// TIA Portal V18 export
FUNCTION_BLOCK "Calculations"   // FB10, LAD
{ S7_Optimized_Access := 'TRUE' }
// stored: AutoNumber false, MemoryReserve 100, SetENOAutomatically false
   VAR
      M1_LPF { S7_SetPoint := 'True'} : "LowPassFilter";
      M2_LPF { S7_SetPoint := 'True'} : "LowPassFilter";
      TDPressFwd_LPF { S7_SetPoint := 'True'} : "LowPassFilter";
      TDPressRev_LPF { S7_SetPoint := 'True'} : "LowPassFilter";
      ClosedLoopTemp_LPF { S7_SetPoint := 'True'} : "LowPassFilter";
      ChargeFlow_LPF { S7_SetPoint := 'True'} : "LowPassFilter";
      HotOilFlow_LPF { S7_SetPoint := 'True'} : "LowPassFilter";
      AuxFlow_LPF { S7_SetPoint := 'True'} : "LowPassFilter";
      ChargePress1_LPF { S7_SetPoint := 'True'} : "LowPassFilter";
      ChargePress2_LPF { S7_SetPoint := 'True'} : "LowPassFilter";
      DrillTorqPotLPF { S7_SetPoint := 'True'} : "LowPassFilter";
      MUTorqPotLPF { S7_SetPoint := 'True'} : "LowPassFilter";
      DrillThrottlePotLPF { S7_SetPoint := 'True'} : "LowPassFilter";
      ActTorq_LPF { S7_SetPoint := 'True'} : "LowPassFilter";
      DrillRecPTO_TP { S7_SetPoint := 'True'} : TP_TIME;
      DrillRecMax { S7_SetPoint := 'True'} : Bool;   // Send max value out to drill recorder
   END_VAR
   VAR_TEMP
      tempReal : Real;
      AutoMUTorqSetLow : Real;
      AutoMUTorqSetHigh : Real;
   END_VAR
   VAR_TEMP   // added for the SCL form of the ladder/FBD networks
      _w1 : Bool;
      _w2 : Bool;
      _w3 : Bool;
      _w4 : Bool;
      _w5 : Bool;
      _w6 : Bool;
   END_VAR
BEGIN

REGION Network 1: Encoder Position
   // Hard coded rollover value to match encoder rollver value from TM Count card
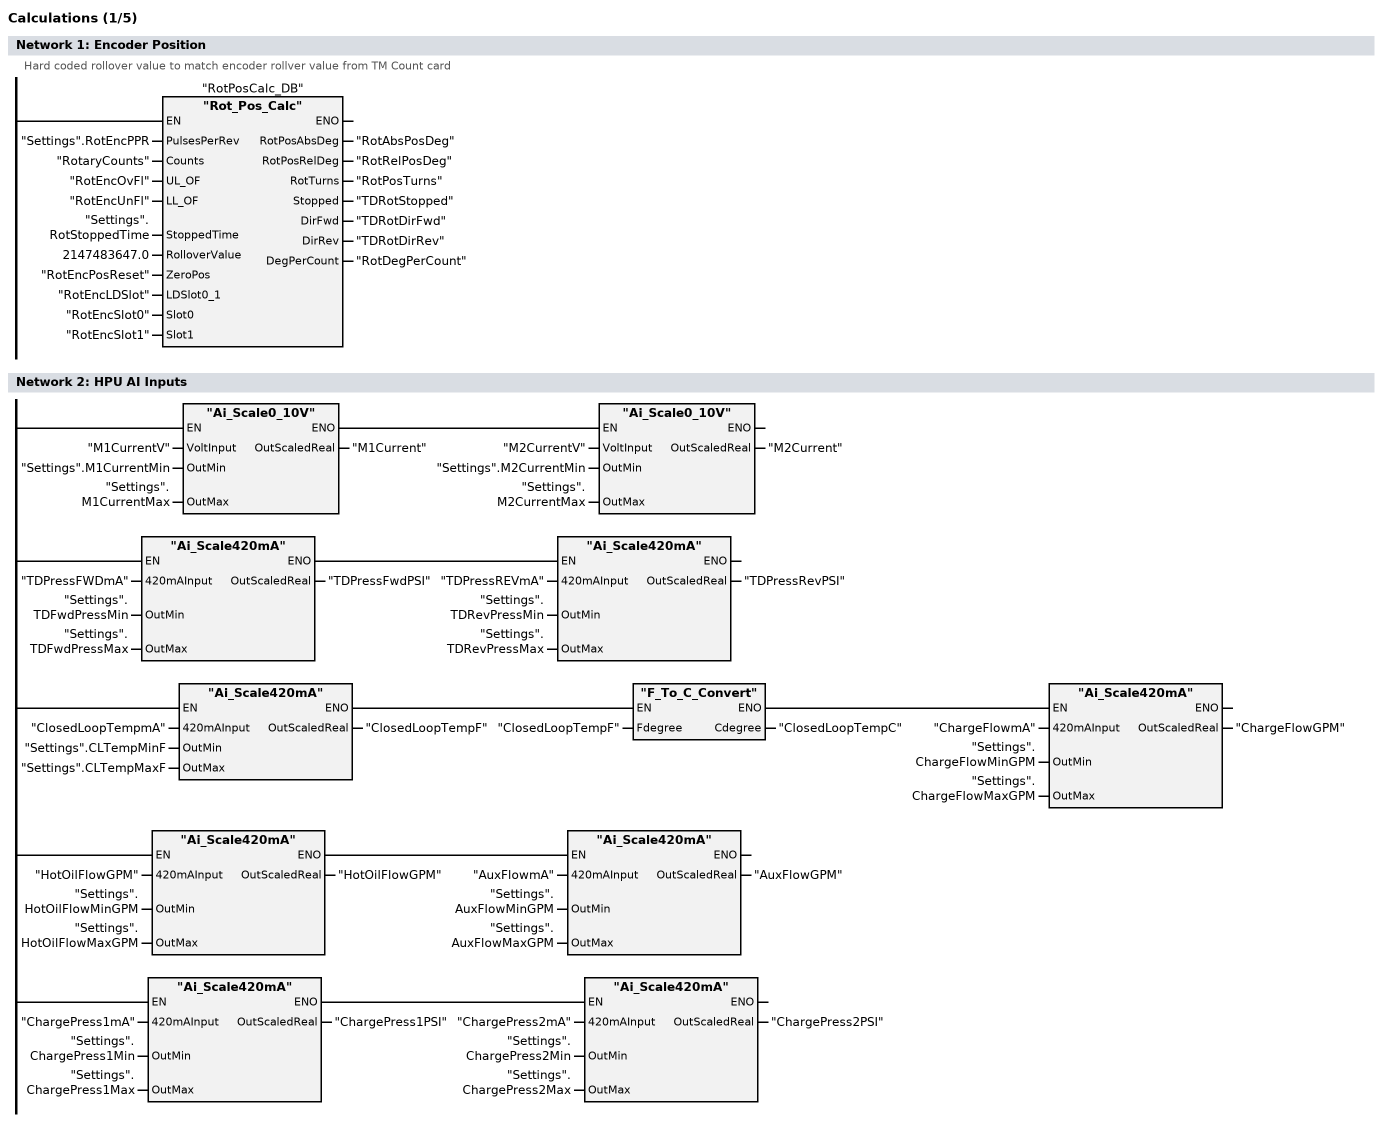
   RUNG wire#powerrail
      "RotPosCalc_DB"(PulsesPerRev := "Settings".RotEncPPR, Counts := "RotaryCounts", UL_OF := "RotEncOvFl", LL_OF := "RotEncUnFl", StoppedTime := "Settings".RotStoppedTime, RolloverValue := 2147483647.0, ZeroPos := "RotEncPosReset", LDSlot0_1 := "RotEncLDSlot", Slot0 := "RotEncSlot0", Slot1 := "RotEncSlot1", RotPosAbsDeg => "RotAbsPosDeg", RotPosRelDeg => "RotRelPosDeg", RotTurns => "RotPosTurns", Stopped => "TDRotStopped", DirFwd => "TDRotDirFwd", DirRev => "TDRotDirRev", DegPerCount => "RotDegPerCount")
   END_RUNG
   // the same network as SCL:
   "RotPosCalc_DB"(PulsesPerRev := "Settings".RotEncPPR,   // "Rot_Pos_Calc"
                   Counts := "RotaryCounts",
                   UL_OF := "RotEncOvFl",
                   LL_OF := "RotEncUnFl",
                   StoppedTime := "Settings".RotStoppedTime,
                   RolloverValue := 2147483647.0,
                   ZeroPos := "RotEncPosReset",
                   LDSlot0_1 := "RotEncLDSlot",
                   Slot0 := "RotEncSlot0",
                   Slot1 := "RotEncSlot1",
                   RotPosAbsDeg => "RotAbsPosDeg",
                   RotPosRelDeg => "RotRelPosDeg",
                   RotTurns => "RotPosTurns",
                   Stopped => "TDRotStopped",
                   DirFwd => "TDRotDirFwd",
                   DirRev => "TDRotDirRev",
                   DegPerCount => "RotDegPerCount");
END_REGION

REGION Network 2: HPU AI Inputs
   RUNG wire#powerrail
      "Ai_Scale0_10V"(VoltInput := "M1CurrentV", OutMin := "Settings".M1CurrentMin, OutMax := "Settings".M1CurrentMax, OutScaledReal => "M1Current")
      "Ai_Scale0_10V"(VoltInput := "M2CurrentV", OutMin := "Settings".M2CurrentMin, OutMax := "Settings".M2CurrentMax, OutScaledReal => "M2Current")
   END_RUNG
   RUNG wire#powerrail
      "Ai_Scale420mA"("420mAInput" := "TDPressFWDmA", OutMin := "Settings".TDFwdPressMin, OutMax := "Settings".TDFwdPressMax, OutScaledReal => "TDPressFwdPSI")
      "Ai_Scale420mA"("420mAInput" := "TDPressREVmA", OutMin := "Settings".TDRevPressMin, OutMax := "Settings".TDRevPressMax, OutScaledReal => "TDPressRevPSI")
   END_RUNG
   RUNG wire#powerrail
      "Ai_Scale420mA"("420mAInput" := "ClosedLoopTempmA", OutMin := "Settings".CLTempMinF, OutMax := "Settings".CLTempMaxF, OutScaledReal => "ClosedLoopTempF")
      "F_To_C_Convert"(Fdegree := "ClosedLoopTempF", Cdegree => "ClosedLoopTempC")
      "Ai_Scale420mA"("420mAInput" := "ChargeFlowmA", OutMin := "Settings".ChargeFlowMinGPM, OutMax := "Settings".ChargeFlowMaxGPM, OutScaledReal => "ChargeFlowGPM")
   END_RUNG
   RUNG wire#powerrail
      "Ai_Scale420mA"("420mAInput" := "HotOilFlowGPM", OutMin := "Settings".HotOilFlowMinGPM, OutMax := "Settings".HotOilFlowMaxGPM, OutScaledReal => "HotOilFlowGPM")
      "Ai_Scale420mA"("420mAInput" := "AuxFlowmA", OutMin := "Settings".AuxFlowMinGPM, OutMax := "Settings".AuxFlowMaxGPM, OutScaledReal => "AuxFlowGPM")
   END_RUNG
   RUNG wire#powerrail
      "Ai_Scale420mA"("420mAInput" := "ChargePress1mA", OutMin := "Settings".ChargePress1Min, OutMax := "Settings".ChargePress1Max, OutScaledReal => "ChargePress1PSI")
      "Ai_Scale420mA"("420mAInput" := "ChargePress2mA", OutMin := "Settings".ChargePress2Min, OutMax := "Settings".ChargePress2Max, OutScaledReal => "ChargePress2PSI")
   END_RUNG
   // the same network as SCL:
   "Ai_Scale0_10V"(VoltInput := "M1CurrentV",
                   OutMin := "Settings".M1CurrentMin,
                   OutMax := "Settings".M1CurrentMax,
                   OutScaledReal => "M1Current",
                   ENO => #_w1);
   IF #_w1 THEN
       "Ai_Scale0_10V"(VoltInput := "M2CurrentV",
                       OutMin := "Settings".M2CurrentMin,
                       OutMax := "Settings".M2CurrentMax,
                       OutScaledReal => "M2Current");
   END_IF;
   "Ai_Scale420mA"("420mAInput" := "TDPressFWDmA",
                   OutMin := "Settings".TDFwdPressMin,
                   OutMax := "Settings".TDFwdPressMax,
                   OutScaledReal => "TDPressFwdPSI",
                   ENO => #_w2);
   IF #_w2 THEN
       "Ai_Scale420mA"("420mAInput" := "TDPressREVmA",
                       OutMin := "Settings".TDRevPressMin,
                       OutMax := "Settings".TDRevPressMax,
                       OutScaledReal => "TDPressRevPSI");
   END_IF;
   "Ai_Scale420mA"("420mAInput" := "ClosedLoopTempmA",
                   OutMin := "Settings".CLTempMinF,
                   OutMax := "Settings".CLTempMaxF,
                   OutScaledReal => "ClosedLoopTempF",
                   ENO => #_w3);
   "F_To_C_Convert"(EN := #_w3, Fdegree := "ClosedLoopTempF", Cdegree => "ClosedLoopTempC", ENO => #_w4);
   IF #_w4 THEN
       "Ai_Scale420mA"("420mAInput" := "ChargeFlowmA",
                       OutMin := "Settings".ChargeFlowMinGPM,
                       OutMax := "Settings".ChargeFlowMaxGPM,
                       OutScaledReal => "ChargeFlowGPM");
   END_IF;
   "Ai_Scale420mA"("420mAInput" := "HotOilFlowGPM",
                   OutMin := "Settings".HotOilFlowMinGPM,
                   OutMax := "Settings".HotOilFlowMaxGPM,
                   OutScaledReal => "HotOilFlowGPM",
                   ENO => #_w5);
   IF #_w5 THEN
       "Ai_Scale420mA"("420mAInput" := "AuxFlowmA",
                       OutMin := "Settings".AuxFlowMinGPM,
                       OutMax := "Settings".AuxFlowMaxGPM,
                       OutScaledReal => "AuxFlowGPM");
   END_IF;
   "Ai_Scale420mA"("420mAInput" := "ChargePress1mA",
                   OutMin := "Settings".ChargePress1Min,
                   OutMax := "Settings".ChargePress1Max,
                   OutScaledReal => "ChargePress1PSI",
                   ENO => #_w6);
   IF #_w6 THEN
       "Ai_Scale420mA"("420mAInput" := "ChargePress2mA",
                       OutMin := "Settings".ChargePress2Min,
                       OutMax := "Settings".ChargePress2Max,
                       OutScaledReal => "ChargePress2PSI");
   END_IF;
END_REGION

REGION Network 3: Filter HPU Inputs
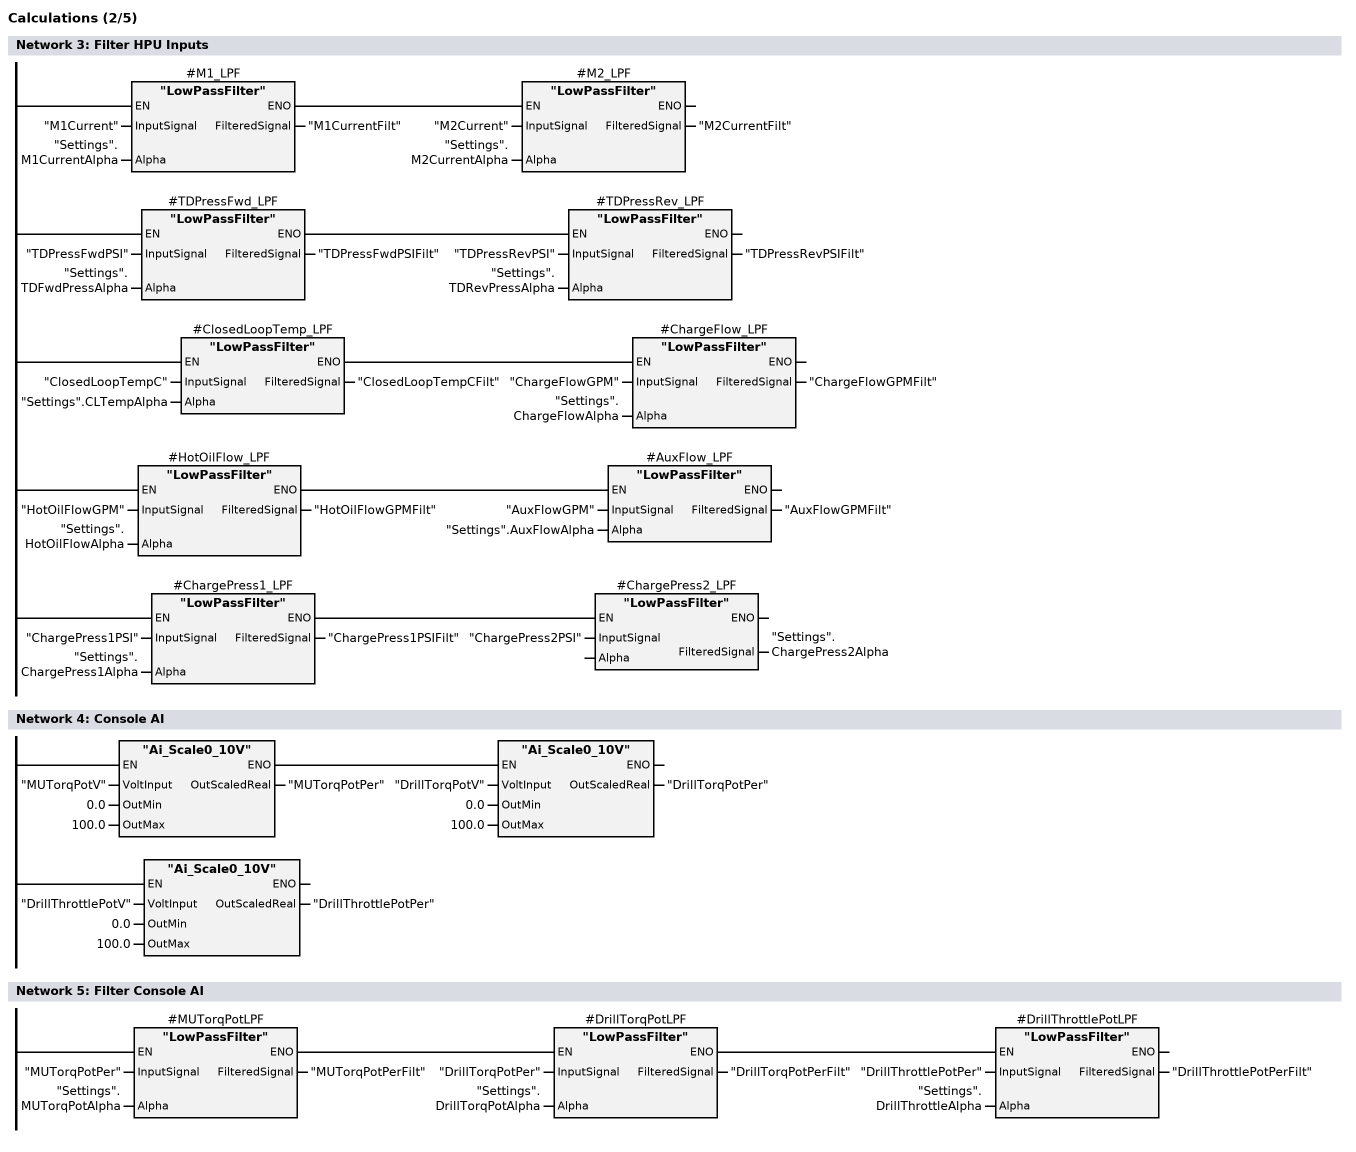
   RUNG wire#powerrail
      #M1_LPF(InputSignal := "M1Current", Alpha := "Settings".M1CurrentAlpha, FilteredSignal => "M1CurrentFilt")
      #M2_LPF(InputSignal := "M2Current", Alpha := "Settings".M2CurrentAlpha, FilteredSignal => "M2CurrentFilt")
   END_RUNG
   RUNG wire#powerrail
      #TDPressFwd_LPF(InputSignal := "TDPressFwdPSI", Alpha := "Settings".TDFwdPressAlpha, FilteredSignal => "TDPressFwdPSIFilt")
      #TDPressRev_LPF(InputSignal := "TDPressRevPSI", Alpha := "Settings".TDRevPressAlpha, FilteredSignal => "TDPressRevPSIFilt")
   END_RUNG
   RUNG wire#powerrail
      #ClosedLoopTemp_LPF(InputSignal := "ClosedLoopTempC", Alpha := "Settings".CLTempAlpha, FilteredSignal => "ClosedLoopTempCFilt")
      #ChargeFlow_LPF(InputSignal := "ChargeFlowGPM", Alpha := "Settings".ChargeFlowAlpha, FilteredSignal => "ChargeFlowGPMFilt")
   END_RUNG
   RUNG wire#powerrail
      #HotOilFlow_LPF(InputSignal := "HotOilFlowGPM", Alpha := "Settings".HotOilFlowAlpha, FilteredSignal => "HotOilFlowGPMFilt")
      #AuxFlow_LPF(InputSignal := "AuxFlowGPM", Alpha := "Settings".AuxFlowAlpha, FilteredSignal => "AuxFlowGPMFilt")
   END_RUNG
   RUNG wire#powerrail
      #ChargePress1_LPF(InputSignal := "ChargePress1PSI", Alpha := "Settings".ChargePress1Alpha, FilteredSignal => "ChargePress1PSIFilt")
      #ChargePress2_LPF(InputSignal := "ChargePress2PSI", Alpha :=, FilteredSignal => "Settings".ChargePress2Alpha)
   END_RUNG
   // the same network as SCL:
   #M1_LPF(InputSignal := "M1Current",   // "LowPassFilter"
           Alpha := "Settings".M1CurrentAlpha,
           FilteredSignal => "M1CurrentFilt",
           ENO => #_w1);
   IF #_w1 THEN
       #M2_LPF(InputSignal := "M2Current", Alpha := "Settings".M2CurrentAlpha, FilteredSignal => "M2CurrentFilt");   // "LowPassFilter"
   END_IF;
   #TDPressFwd_LPF(InputSignal := "TDPressFwdPSI",   // "LowPassFilter"
                   Alpha := "Settings".TDFwdPressAlpha,
                   FilteredSignal => "TDPressFwdPSIFilt",
                   ENO => #_w2);
   IF #_w2 THEN
       #TDPressRev_LPF(InputSignal := "TDPressRevPSI",   // "LowPassFilter"
                       Alpha := "Settings".TDRevPressAlpha,
                       FilteredSignal => "TDPressRevPSIFilt");
   END_IF;
   #ClosedLoopTemp_LPF(InputSignal := "ClosedLoopTempC",   // "LowPassFilter"
                       Alpha := "Settings".CLTempAlpha,
                       FilteredSignal => "ClosedLoopTempCFilt",
                       ENO => #_w3);
   IF #_w3 THEN
       #ChargeFlow_LPF(InputSignal := "ChargeFlowGPM",   // "LowPassFilter"
                       Alpha := "Settings".ChargeFlowAlpha,
                       FilteredSignal => "ChargeFlowGPMFilt");
   END_IF;
   #HotOilFlow_LPF(InputSignal := "HotOilFlowGPM",   // "LowPassFilter"
                   Alpha := "Settings".HotOilFlowAlpha,
                   FilteredSignal => "HotOilFlowGPMFilt",
                   ENO => #_w4);
   IF #_w4 THEN
       #AuxFlow_LPF(InputSignal := "AuxFlowGPM",   // "LowPassFilter"
                    Alpha := "Settings".AuxFlowAlpha,
                    FilteredSignal => "AuxFlowGPMFilt");
   END_IF;
   #ChargePress1_LPF(InputSignal := "ChargePress1PSI",   // "LowPassFilter"
                     Alpha := "Settings".ChargePress1Alpha,
                     FilteredSignal => "ChargePress1PSIFilt",
                     ENO => #_w5);
   IF #_w5 THEN
       #ChargePress2_LPF(InputSignal := "ChargePress2PSI", FilteredSignal => "Settings".ChargePress2Alpha);   // "LowPassFilter"
   END_IF;
END_REGION

REGION Network 4: Console AI
   RUNG wire#powerrail
      "Ai_Scale0_10V"(VoltInput := "MUTorqPotV", OutMin := 0.0, OutMax := 100.0, OutScaledReal => "MUTorqPotPer")
      "Ai_Scale0_10V"(VoltInput := "DrillTorqPotV", OutMin := 0.0, OutMax := 100.0, OutScaledReal => "DrillTorqPotPer")
   END_RUNG
   RUNG wire#powerrail
      "Ai_Scale0_10V"(VoltInput := "DrillThrottlePotV", OutMin := 0.0, OutMax := 100.0, OutScaledReal => "DrillThrottlePotPer")
   END_RUNG
   // the same network as SCL:
   "Ai_Scale0_10V"(VoltInput := "MUTorqPotV",
                   OutMin := 0.0,
                   OutMax := 100.0,
                   OutScaledReal => "MUTorqPotPer",
                   ENO => #_w1);
   IF #_w1 THEN
       "Ai_Scale0_10V"(VoltInput := "DrillTorqPotV",
                       OutMin := 0.0,
                       OutMax := 100.0,
                       OutScaledReal => "DrillTorqPotPer");
   END_IF;
   "Ai_Scale0_10V"(VoltInput := "DrillThrottlePotV",
                   OutMin := 0.0,
                   OutMax := 100.0,
                   OutScaledReal => "DrillThrottlePotPer");
END_REGION

REGION Network 5: Filter Console AI
   RUNG wire#powerrail
      #MUTorqPotLPF(InputSignal := "MUTorqPotPer", Alpha := "Settings".MUTorqPotAlpha, FilteredSignal => "MUTorqPotPerFilt")
      #DrillTorqPotLPF(InputSignal := "DrillTorqPotPer", Alpha := "Settings".DrillTorqPotAlpha, FilteredSignal => "DrillTorqPotPerFilt")
      #DrillThrottlePotLPF(InputSignal := "DrillThrottlePotPer", Alpha := "Settings".DrillThrottleAlpha, FilteredSignal => "DrillThrottlePotPerFilt")
   END_RUNG
   // the same network as SCL:
   #MUTorqPotLPF(InputSignal := "MUTorqPotPer",   // "LowPassFilter"
                 Alpha := "Settings".MUTorqPotAlpha,
                 FilteredSignal => "MUTorqPotPerFilt",
                 ENO => #_w1);
   #DrillTorqPotLPF(EN := #_w1,   // "LowPassFilter"
                    InputSignal := "DrillTorqPotPer",
                    Alpha := "Settings".DrillTorqPotAlpha,
                    FilteredSignal => "DrillTorqPotPerFilt",
                    ENO => #_w2);
   IF #_w2 THEN
       #DrillThrottlePotLPF(InputSignal := "DrillThrottlePotPer",   // "LowPassFilter"
                            Alpha := "Settings".DrillThrottleAlpha,
                            FilteredSignal => "DrillThrottlePotPerFilt");
   END_IF;
END_REGION

REGION Network 6: Torque Calculation
   // Differential Pressure x torque factor(ft-lbs/psi) unless bypass running * efficiency. Use raw reading value and filter after
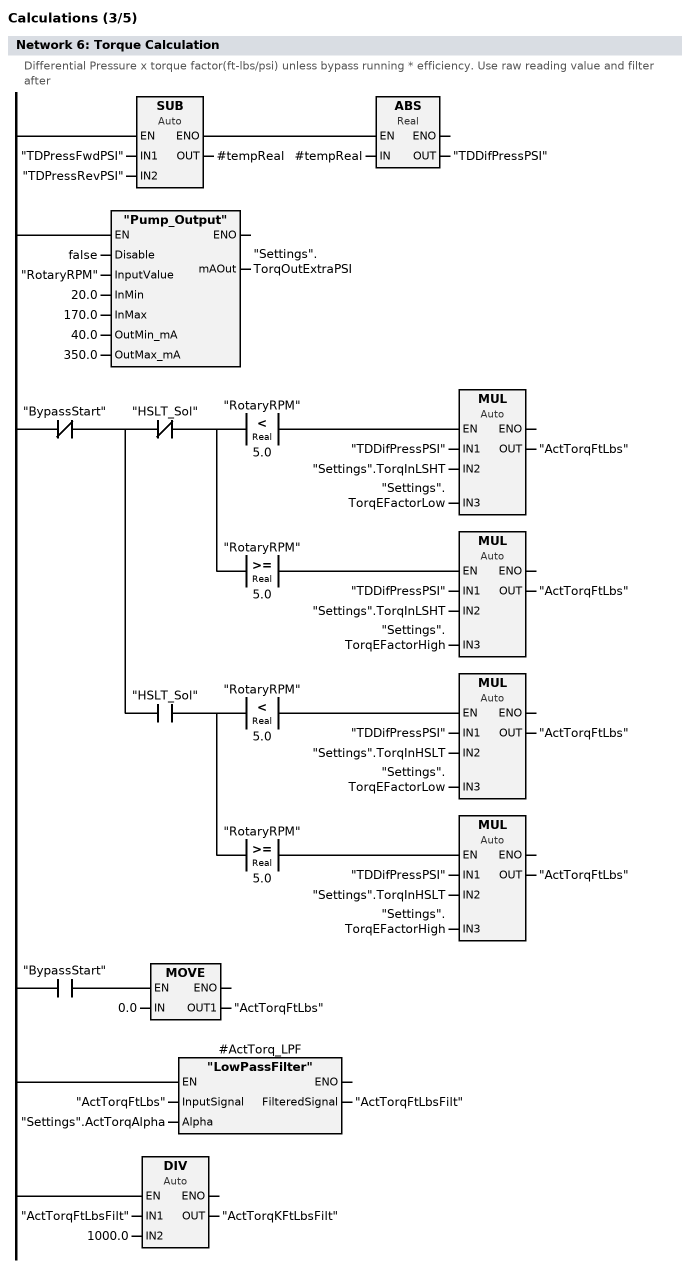
   RUNG wire#powerrail
      Sub(in1 := "TDPressFwdPSI", in2 := "TDPressRevPSI", out => #tempReal)
      { S7_Templates := "SrcType := Real" } Abs(in := #tempReal, out => "TDDifPressPSI")
   END_RUNG
   RUNG wire#powerrail
      "Pump_Output"(Disable := false, InputValue := "RotaryRPM", InMin := 20.0, InMax := 170.0, OutMin_mA := 40.0, OutMax_mA := 350.0, mAOut => "Settings".TorqOutExtraPSI)
   END_RUNG
   RUNG wire#powerrail
      I_Contact( "BypassStart" )
      wire#w1
      I_Contact( "HSLT_Sol" )
      wire#w2
      { S7_Templates := "SrcType := Real" } LT_Contact(in1 := "RotaryRPM", in2 := 5.0)
      Mul(in1 := "TDDifPressPSI", in2 := "Settings".TorqInLSHT, in3 := "Settings".TorqEFactorLow, out => "ActTorqFtLbs")
   END_RUNG
   RUNG wire#w2
      { S7_Templates := "SrcType := Real" } GE_Contact(in1 := "RotaryRPM", in2 := 5.0)
      Mul(in1 := "TDDifPressPSI", in2 := "Settings".TorqInLSHT, in3 := "Settings".TorqEFactorHigh, out => "ActTorqFtLbs")
   END_RUNG
   RUNG wire#w1
      Contact( "HSLT_Sol" )
      wire#w3
      { S7_Templates := "SrcType := Real" } LT_Contact(in1 := "RotaryRPM", in2 := 5.0)
      Mul(in1 := "TDDifPressPSI", in2 := "Settings".TorqInHSLT, in3 := "Settings".TorqEFactorLow, out => "ActTorqFtLbs")
   END_RUNG
   RUNG wire#w3
      { S7_Templates := "SrcType := Real" } GE_Contact(in1 := "RotaryRPM", in2 := 5.0)
      Mul(in1 := "TDDifPressPSI", in2 := "Settings".TorqInHSLT, in3 := "Settings".TorqEFactorHigh, out => "ActTorqFtLbs")
   END_RUNG
   RUNG wire#powerrail
      Contact( "BypassStart" )
      Move(in := 0.0, out1 => "ActTorqFtLbs")
   END_RUNG
   RUNG wire#powerrail
      #ActTorq_LPF(InputSignal := "ActTorqFtLbs", Alpha := "Settings".ActTorqAlpha, FilteredSignal => "ActTorqFtLbsFilt")
   END_RUNG
   RUNG wire#powerrail
      Div(in1 := "ActTorqFtLbsFilt", in2 := 1000.0, out => "ActTorqKFtLbsFilt")
   END_RUNG
   // the same network as SCL:
   #tempReal := "TDPressFwdPSI" - "TDPressRevPSI";
   "TDDifPressPSI" := ABS(#tempReal);
   "Pump_Output"(Disable := false,
                 InputValue := "RotaryRPM",
                 InMin := 20.0,
                 InMax := 170.0,
                 OutMin_mA := 40.0,
                 OutMax_mA := 350.0,
                 mAOut => "Settings".TorqOutExtraPSI);
   #_w1 := NOT "BypassStart" AND NOT "HSLT_Sol";
   IF #_w1 AND ("RotaryRPM" < 5.0) THEN
       "ActTorqFtLbs" := "TDDifPressPSI" * "Settings".TorqInLSHT * "Settings".TorqEFactorLow;
   END_IF;
   IF #_w1 AND ("RotaryRPM" >= 5.0) THEN
       "ActTorqFtLbs" := "TDDifPressPSI" * "Settings".TorqInLSHT * "Settings".TorqEFactorHigh;
   END_IF;
   #_w2 := NOT "BypassStart" AND "HSLT_Sol";
   IF #_w2 AND ("RotaryRPM" < 5.0) THEN
       "ActTorqFtLbs" := "TDDifPressPSI" * "Settings".TorqInHSLT * "Settings".TorqEFactorLow;
   END_IF;
   IF #_w2 AND ("RotaryRPM" >= 5.0) THEN
       "ActTorqFtLbs" := "TDDifPressPSI" * "Settings".TorqInHSLT * "Settings".TorqEFactorHigh;
   END_IF;
   IF "BypassStart" THEN "ActTorqFtLbs" := 0.0; END_IF;
   #ActTorq_LPF(InputSignal := "ActTorqFtLbs",   // "LowPassFilter"
                Alpha := "Settings".ActTorqAlpha,
                FilteredSignal => "ActTorqFtLbsFilt");
   "ActTorqKFtLbsFilt" := "ActTorqFtLbsFilt" / 1000.0;
END_REGION

REGION Network 7: User Setpoints
   // Drill torque setpoint cannot be greater than 0.95 % of the makeup setpoint
   // MU Torque always low speed as it cannot shift
   // Drill torque depends on speed settings
   // MU threshold is a percent of setpoint
   // Add 500 PSI to setpoint to overcome charge pressure
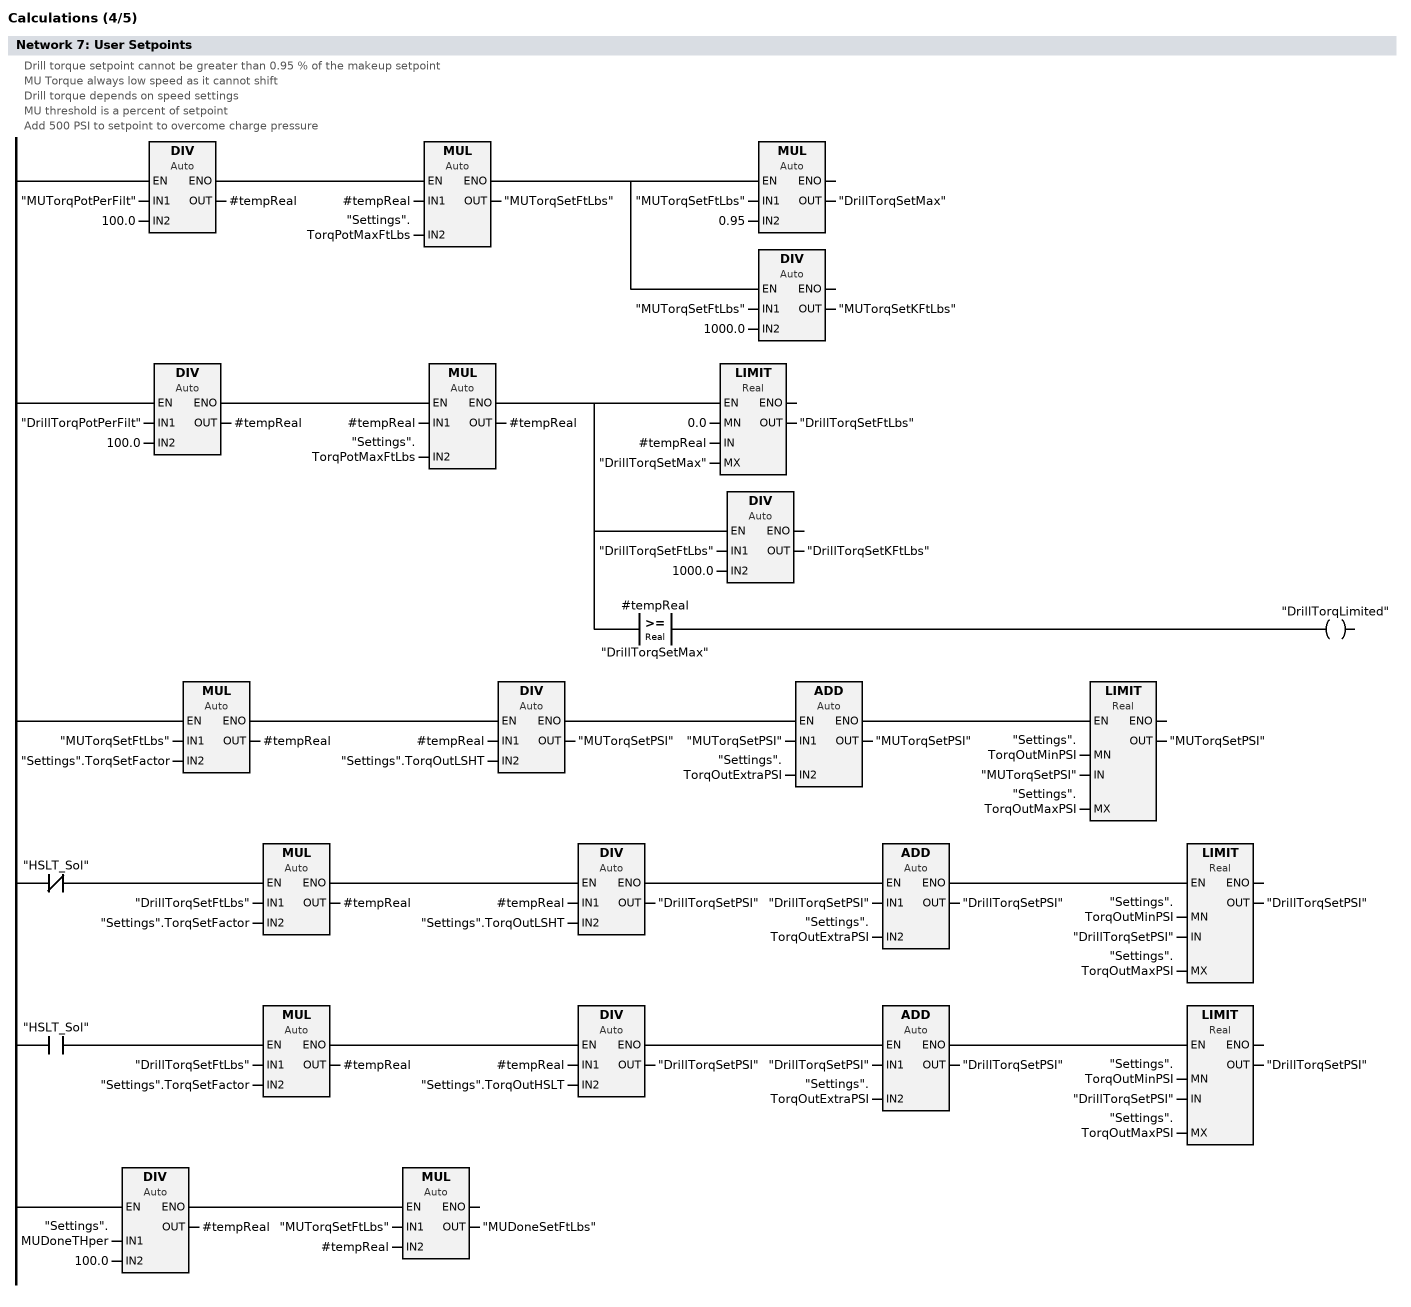
   RUNG wire#powerrail
      Div(in1 := "MUTorqPotPerFilt", in2 := 100.0, out => #tempReal)
      Mul(in1 := #tempReal, in2 := "Settings".TorqPotMaxFtLbs, out => "MUTorqSetFtLbs")
      wire#w1
      Mul(in1 := "MUTorqSetFtLbs", in2 := 0.95, out => "DrillTorqSetMax")
   END_RUNG
   RUNG wire#w1
      Div(in1 := "MUTorqSetFtLbs", in2 := 1000.0, out => "MUTorqSetKFtLbs")
   END_RUNG
   RUNG wire#powerrail
      Div(in1 := "DrillTorqPotPerFilt", in2 := 100.0, out => #tempReal)
      Mul(in1 := #tempReal, in2 := "Settings".TorqPotMaxFtLbs, out => #tempReal)
      wire#w2
      { S7_Templates := "value_type := Real" } Limit(mn := 0.0, in := #tempReal, mx := "DrillTorqSetMax", out => "DrillTorqSetFtLbs")
   END_RUNG
   RUNG wire#w2
      Div(in1 := "DrillTorqSetFtLbs", in2 := 1000.0, out => "DrillTorqSetKFtLbs")
   END_RUNG
   RUNG wire#w2
      { S7_Templates := "SrcType := Real" } GE_Contact(in1 := #tempReal, in2 := "DrillTorqSetMax")
      Coil( "DrillTorqLimited" )
   END_RUNG
   RUNG wire#powerrail
      Mul(in1 := "MUTorqSetFtLbs", in2 := "Settings".TorqSetFactor, out => #tempReal)
      Div(in1 := #tempReal, in2 := "Settings".TorqOutLSHT, out => "MUTorqSetPSI")
      Add(in1 := "MUTorqSetPSI", in2 := "Settings".TorqOutExtraPSI, out => "MUTorqSetPSI")
      { S7_Templates := "value_type := Real" } Limit(mn := "Settings".TorqOutMinPSI, in := "MUTorqSetPSI", mx := "Settings".TorqOutMaxPSI, out => "MUTorqSetPSI")
   END_RUNG
   RUNG wire#powerrail
      I_Contact( "HSLT_Sol" )
      Mul(in1 := "DrillTorqSetFtLbs", in2 := "Settings".TorqSetFactor, out => #tempReal)
      Div(in1 := #tempReal, in2 := "Settings".TorqOutLSHT, out => "DrillTorqSetPSI")
      Add(in1 := "DrillTorqSetPSI", in2 := "Settings".TorqOutExtraPSI, out => "DrillTorqSetPSI")
      { S7_Templates := "value_type := Real" } Limit(mn := "Settings".TorqOutMinPSI, in := "DrillTorqSetPSI", mx := "Settings".TorqOutMaxPSI, out => "DrillTorqSetPSI")
   END_RUNG
   RUNG wire#powerrail
      Contact( "HSLT_Sol" )
      Mul(in1 := "DrillTorqSetFtLbs", in2 := "Settings".TorqSetFactor, out => #tempReal)
      Div(in1 := #tempReal, in2 := "Settings".TorqOutHSLT, out => "DrillTorqSetPSI")
      Add(in1 := "DrillTorqSetPSI", in2 := "Settings".TorqOutExtraPSI, out => "DrillTorqSetPSI")
      { S7_Templates := "value_type := Real" } Limit(mn := "Settings".TorqOutMinPSI, in := "DrillTorqSetPSI", mx := "Settings".TorqOutMaxPSI, out => "DrillTorqSetPSI")
   END_RUNG
   RUNG wire#powerrail
      Div(in1 := "Settings".MUDoneTHper, in2 := 100.0, out => #tempReal)
      Mul(in1 := "MUTorqSetFtLbs", in2 := #tempReal, out => "MUDoneSetFtLbs")
   END_RUNG
   // the same network as SCL:
   #tempReal := "MUTorqPotPerFilt" / 100.0;
   "MUTorqSetFtLbs" := #tempReal * "Settings".TorqPotMaxFtLbs;
   "DrillTorqSetMax" := "MUTorqSetFtLbs" * 0.95;
   "MUTorqSetKFtLbs" := "MUTorqSetFtLbs" / 1000.0;
   #tempReal := "DrillTorqPotPerFilt" / 100.0;
   #tempReal := #tempReal * "Settings".TorqPotMaxFtLbs;
   "DrillTorqSetFtLbs" := LIMIT(MN := 0.0, IN := #tempReal, MX := "DrillTorqSetMax");
   "DrillTorqSetKFtLbs" := "DrillTorqSetFtLbs" / 1000.0;
   "DrillTorqLimited" := #tempReal >= "DrillTorqSetMax";
   #tempReal := "MUTorqSetFtLbs" * "Settings".TorqSetFactor;
   "MUTorqSetPSI" := #tempReal / "Settings".TorqOutLSHT;
   "MUTorqSetPSI" := "MUTorqSetPSI" + "Settings".TorqOutExtraPSI;
   "MUTorqSetPSI" := LIMIT(MN := "Settings".TorqOutMinPSI, IN := "MUTorqSetPSI", MX := "Settings".TorqOutMaxPSI);
   IF NOT "HSLT_Sol" THEN
       #tempReal := "DrillTorqSetFtLbs" * "Settings".TorqSetFactor;
       "DrillTorqSetPSI" := #tempReal / "Settings".TorqOutLSHT;
       "DrillTorqSetPSI" := "DrillTorqSetPSI" + "Settings".TorqOutExtraPSI;
       "DrillTorqSetPSI" := LIMIT(MN := "Settings".TorqOutMinPSI, IN := "DrillTorqSetPSI", MX := "Settings".TorqOutMaxPSI);
   END_IF;
   IF "HSLT_Sol" THEN
       #tempReal := "DrillTorqSetFtLbs" * "Settings".TorqSetFactor;
       "DrillTorqSetPSI" := #tempReal / "Settings".TorqOutHSLT;
       "DrillTorqSetPSI" := "DrillTorqSetPSI" + "Settings".TorqOutExtraPSI;
       "DrillTorqSetPSI" := LIMIT(MN := "Settings".TorqOutMinPSI, IN := "DrillTorqSetPSI", MX := "Settings".TorqOutMaxPSI);
   END_IF;
   #tempReal := "Settings".MUDoneTHper / 100.0;
   "MUDoneSetFtLbs" := "MUTorqSetFtLbs" * #tempReal;
END_REGION

REGION Network 8: Auto Makeup Torq Setpoints
   // These setpoints are based on a percent of the user input
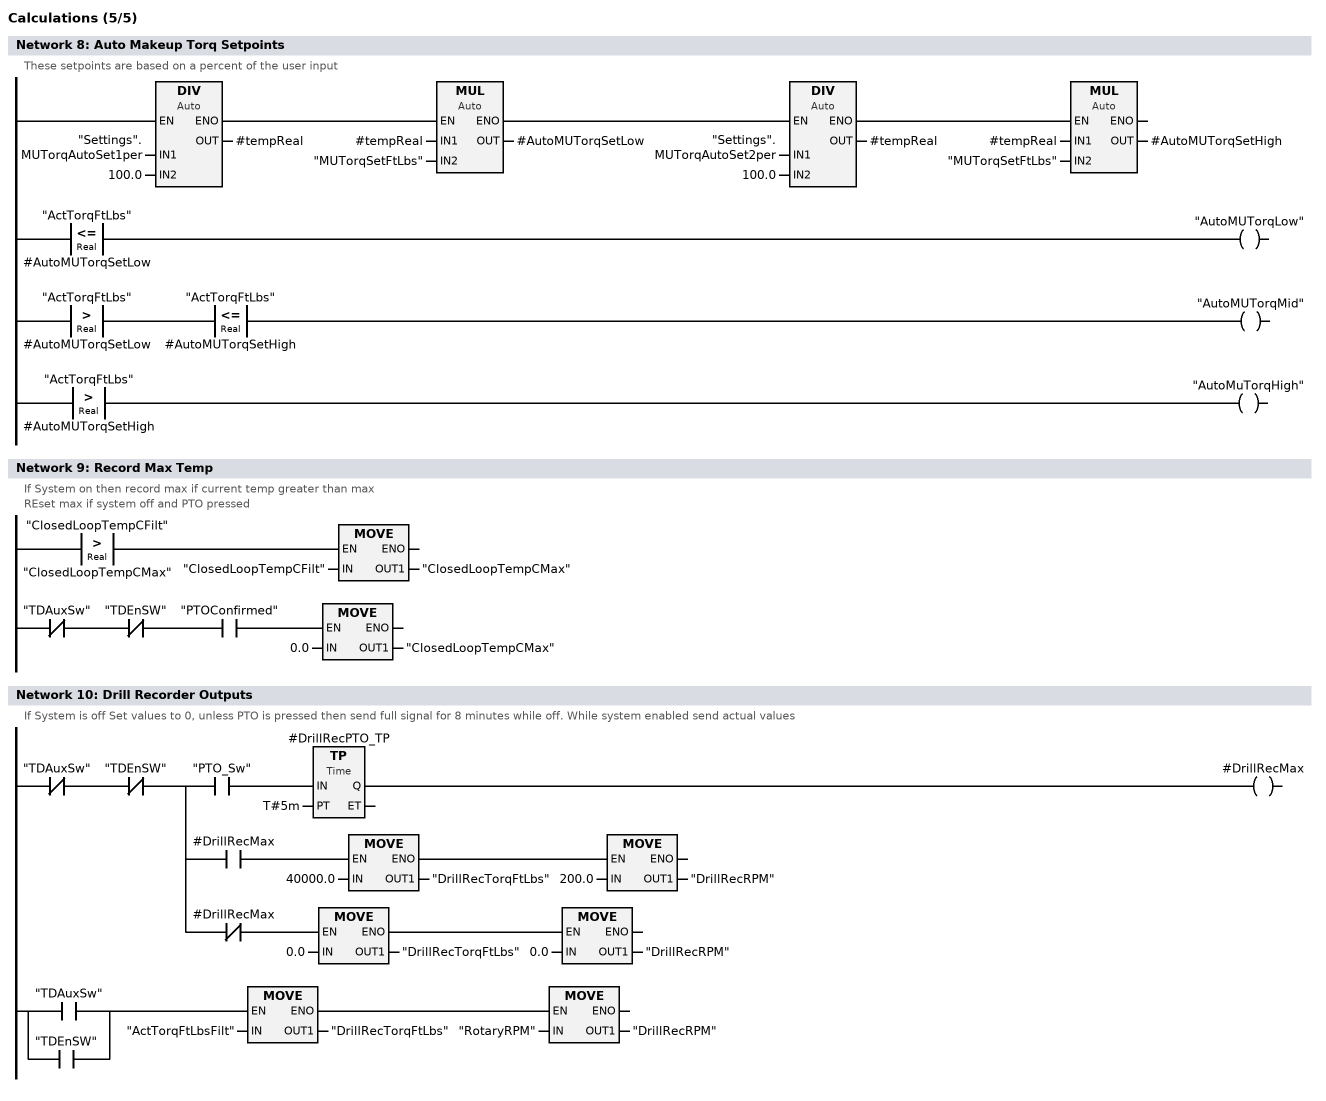
   RUNG wire#powerrail
      Div(in1 := "Settings".MUTorqAutoSet1per, in2 := 100.0, out => #tempReal)
      Mul(in1 := #tempReal, in2 := "MUTorqSetFtLbs", out => #AutoMUTorqSetLow)
      Div(in1 := "Settings".MUTorqAutoSet2per, in2 := 100.0, out => #tempReal)
      Mul(in1 := #tempReal, in2 := "MUTorqSetFtLbs", out => #AutoMUTorqSetHigh)
   END_RUNG
   RUNG wire#powerrail
      { S7_Templates := "SrcType := Real" } LE_Contact(in1 := "ActTorqFtLbs", in2 := #AutoMUTorqSetLow)
      Coil( "AutoMUTorqLow" )
   END_RUNG
   RUNG wire#powerrail
      { S7_Templates := "SrcType := Real" } GT_Contact(in1 := "ActTorqFtLbs", in2 := #AutoMUTorqSetLow)
      { S7_Templates := "SrcType := Real" } LE_Contact(in1 := "ActTorqFtLbs", in2 := #AutoMUTorqSetHigh)
      Coil( "AutoMUTorqMid" )
   END_RUNG
   RUNG wire#powerrail
      { S7_Templates := "SrcType := Real" } GT_Contact(in1 := "ActTorqFtLbs", in2 := #AutoMUTorqSetHigh)
      Coil( "AutoMuTorqHigh" )
   END_RUNG
   // the same network as SCL:
   #tempReal := "Settings".MUTorqAutoSet1per / 100.0;
   #AutoMUTorqSetLow := #tempReal * "MUTorqSetFtLbs";
   #tempReal := "Settings".MUTorqAutoSet2per / 100.0;
   #AutoMUTorqSetHigh := #tempReal * "MUTorqSetFtLbs";
   "AutoMUTorqLow" := "ActTorqFtLbs" <= #AutoMUTorqSetLow;
   "AutoMUTorqMid" := ("ActTorqFtLbs" > #AutoMUTorqSetLow) AND ("ActTorqFtLbs" <= #AutoMUTorqSetHigh);
   "AutoMuTorqHigh" := "ActTorqFtLbs" > #AutoMUTorqSetHigh;
END_REGION

REGION Network 9: Record Max Temp
   // If System on then record max if current temp greater than max
   // REset max if system off and PTO pressed
   RUNG wire#powerrail
      { S7_Templates := "SrcType := Real" } GT_Contact(in1 := "ClosedLoopTempCFilt", in2 := "ClosedLoopTempCMax")
      Move(in := "ClosedLoopTempCFilt", out1 => "ClosedLoopTempCMax")
   END_RUNG
   RUNG wire#powerrail
      I_Contact( "TDAuxSw" )
      I_Contact( "TDEnSW" )
      Contact( "PTOConfirmed" )
      Move(in := 0.0, out1 => "ClosedLoopTempCMax")
   END_RUNG
   // the same network as SCL:
   IF "ClosedLoopTempCFilt" > "ClosedLoopTempCMax" THEN
       "ClosedLoopTempCMax" := "ClosedLoopTempCFilt";
   END_IF;
   IF NOT "TDAuxSw" AND NOT "TDEnSW" AND "PTOConfirmed" THEN "ClosedLoopTempCMax" := 0.0; END_IF;
END_REGION

REGION Network 10: Drill Recorder Outputs
   // If System is off Set values to 0, unless PTO is pressed then send full signal for 8 minutes while off. While system enabled send actual values
   RUNG wire#powerrail
      I_Contact( "TDAuxSw" )
      I_Contact( "TDEnSW" )
      wire#w1
      Contact( "PTO_Sw" )
      { S7_Templates := "time_type := Time" } #DrillRecPTO_TP.TP(pt := T#5m, et =>)
      Coil( #DrillRecMax )
   END_RUNG
   RUNG wire#w1
      Contact( #DrillRecMax )
      Move(in := 40000.0, out1 => "DrillRecTorqFtLbs")
      Move(in := 200.0, out1 => "DrillRecRPM")
   END_RUNG
   RUNG wire#w1
      I_Contact( #DrillRecMax )
      Move(in := 0.0, out1 => "DrillRecTorqFtLbs")
      Move(in := 0.0, out1 => "DrillRecRPM")
   END_RUNG
   RUNG wire#powerrail
      Contact( "TDAuxSw" )
      wire#w2
      Move(in := "ActTorqFtLbsFilt", out1 => "DrillRecTorqFtLbs")
      Move(in := "RotaryRPM", out1 => "DrillRecRPM")
   END_RUNG
   RUNG wire#powerrail
      Contact( "TDEnSW" )
   END_RUNG wire#w2
   // the same network as SCL:
   #_w1 := NOT "TDAuxSw" AND NOT "TDEnSW";
   #DrillRecPTO_TP(IN := #_w1 AND "PTO_Sw", PT := T#5m);   // TP
   #DrillRecMax := #DrillRecPTO_TP.Q;
   IF #_w1 AND #DrillRecMax THEN
       "DrillRecTorqFtLbs" := 40000.0;
       "DrillRecRPM" := 200.0;
   END_IF;
   IF #_w1 AND NOT #DrillRecMax THEN
       "DrillRecTorqFtLbs" := 0.0;
       "DrillRecRPM" := 0.0;
   END_IF;
   IF "TDAuxSw" OR "TDEnSW" THEN
       "DrillRecTorqFtLbs" := "ActTorqFtLbsFilt";
       "DrillRecRPM" := "RotaryRPM";
   END_IF;
END_REGION
END_FUNCTION_BLOCK
